// TwinCAT 3 PLC project PLC1
// ProgramVersion: 3.1.4024.12
// libraries:
//   Tc2_Standard, * (Beckhoff Automation GmbH)
//   Tc2_System, * (Beckhoff Automation GmbH)
//   Tc3_Module, * (Beckhoff Automation GmbH)
// project tree:
//   Diagrams/ Class Diagram.TcCD (not stored)
//   FBs/ FB_LAMP_DIAG.TcPOU, FB_LAMP_DIMM.TcPOU, FB_LAMP_ONOFF.TcPOU (not stored)
//   Git/Gi1/ Git1_FB.TcPOU
//   Git/Git2/ Git2_FB.TcPOU
//   ITFs/ I_LampCtrl.TcIO (not stored), I_LampCtrl_Diag.TcIO
//   / PlcTask.TcTTO (not stored)
//   POUs/ MAIN.TcPOU
// real-time tasks:
//   TASK PlcTask: cycle T#10ms, priority 20, ADS port 350

// ---- ITFs/I_LampCtrl_Diag.TcIO
INTERFACE I_LampCtrl_Diag EXTENDS I_LampCtrl

METHOD CheckLampID : INT
VAR_INPUT
	I_xStart	:	BOOL;
END_VAR
END_METHOD

METHOD Diag : BOOL
END_METHOD

END_INTERFACE

// ---- FBs/FB_LAMP_DIAG.TcPOU
FUNCTION_BLOCK FB_LAMP_DIAG EXTENDS FB_LAMP_ONOFF IMPLEMENTS I_LampCtrl_Diag;
VAR_INPUT
END_VAR
VAR_OUTPUT
END_VAR
VAR
	xSN							: INT;
	iInTemperatureHw	AT %I*	: INT;
END_VAR

METHOD CheckLampID : INT
VAR_INPUT
	I_xStart	:	BOOL;
END_VAR
IF I_xStart THEN
	CheckLampID	:= xSN;
END_IF
END_METHOD

METHOD Diag : BOOL
Diag := FALSE;

IF iInTemperatureHw > 200 THEN
	SUPER^.OFF();
END_IF

DIAG := TRUE;
END_METHOD

END_FUNCTION_BLOCK

// ---- FBs/FB_LAMP_DIMM.TcPOU
{attribute 'reflection'}
FUNCTION_BLOCK FB_LAMP_DIMM IMPLEMENTS I_LampCtrl
VAR_INPUT
END_VAR
VAR_OUTPUT
END_VAR
VAR
	
	fOut :REAL;
	fInc :REAL:=0.5;
	iOutHw AT%Q*:INT; // Output to Dimmer
	
	{attribute 'instance-path'}
	{attribute 'no_init'}
	sPath: STRING;
END_VAR

METHOD OFF : BOOL
// implementation dimm++. 
//Intensity in 0..100%  variable fOut 
fOut :=fOut - fInc;
IF fOut < 0.0 THEN
    fOut :=0.0;
	OFF := TRUE;
ELSE
	OFF := FALSE;
END_IF

// conversion to hardware output 0..32767
iOutHw := LIMIT (0,REAL_TO_INT(fOut * 32.767),32767); // for dimmer output
END_METHOD

METHOD ON : BOOL
// implementation dimm++. 
//Intensity in 0..100%  variable fOut 
fOut :=fOut + fInc;
IF fOut > 100.0 THEN
    fOut :=100.0;
	On := TRUE;
ELSE
	On := FALSE;
END_IF
iOutHw := LIMIT (0,REAL_TO_INT(fOut * 327.67),32767); // for dimmer output
END_METHOD

PROPERTY State : string
GET
State := CONCAT('Object:', sPath); 
State := CONCAT(State, 'State (%):'); 
State := CONCAT(State, REAL_TO_STRING(fOut));
END_GET
END_PROPERTY

END_FUNCTION_BLOCK

// ---- Git/Gi1/Git1_FB.TcPOU
FUNCTION_BLOCK Git1_FB
VAR_INPUT
END_VAR
VAR_OUTPUT
END_VAR
VAR
END_VAR

END_FUNCTION_BLOCK

// ---- Git/Git2/Git2_FB.TcPOU
FUNCTION_BLOCK Git2_FB
VAR_INPUT
END_VAR
VAR_OUTPUT
END_VAR
VAR
END_VAR

END_FUNCTION_BLOCK

// ---- POUs/MAIN.TcPOU
PROGRAM MAIN
VAR
	// Used to demo ITF reference on start-up
	fbLamp1 	: FB_LAMP_DIMM;
	fbLamp2 	: FB_LAMP_ONOFF;
	fbLampDiag	: FB_LAMP_DIAG;
	fbLampDiag2	: FB_LAMP_DIAG;
	
	// Interface
	LampCtrl 	: ARRAY[0..2] OF I_LampCtrl := [fbLamp1, fbLamp2, fbLampDiag2];
	ILampCtrl_Diag :	I_LampCtrl_Diag := fbLampDiag;
	
	// Program Control
	bLightsOn	: BOOL;
	bLightsOff	: BOOL;
	State		: ARRAY[0..1] OF STRING;
	eRet		: INT;
END_VAR

IF bLightsOn THEN
	IF LampCtrl[0].ON() AND LampCtrl[1].ON() THEN
		bLightsOn := FALSE;
	END_IF
END_IF

IF bLightsOff THEN	
	IF LampCtrl[0].OFF() AND LampCtrl[1].OFF() THEN
		bLightsOff := FALSE;
	END_IF
END_IF

LampCtrl[2].OFF();

State[0] := LampCtrl[0].State;
State[1] := LampCtrl[1].State;

eRet	:=	ILampCtrl_Diag.CheckLampID(I_xStart := TRUE);

END_PROGRAM
